FUNCTION_BLOCK PICKUP_SCREW
VAR_INPUT
END_VAR
VAR_OUTPUT
END_VAR
VAR
END_VAR

END_FUNCTION_BLOCK

(* stored: Version 1.1.0.1, ProductVersion 3.1.4022.18
   POU PICKUP_SCREW: Id {99d35285-e01c-443f-8d46-44984eaa44c8}, SpecialFunc None *)
